// TIA Portal V19 export
DATA_BLOCK "AreaGen_Msg_Alarms"   // DB181
// stored: InstanceOfName MsgManager, InstanceOfType FB
"MsgManager"
   // VAR_INPUT
   //    Ack : Bool;
   // END_VAR
   // VAR_OUTPUT
   //    MessagePresence : Bool;
   //    NewMessage : Bool;
   //    MessageCount : Int;
   // END_VAR
   // VAR_IN_OUT
   //    Messages : Array[*] of Bool;
   //    MessagesHMI : Array[*] of Word;
   //    MessagesACK : Array[*] of Word;
   // END_VAR
   // VAR
   //    MsgDim : DInt;
   //    HmiMsgDim : DInt;
   //    AckMsgDim : DInt;
   //    MsgCount : Int;
   //    Status : Int;
   //    IndexBuild : Int;
   //    IndexCompare : Int;
   //    LoopStart : Int;
   //    LoopEnd : Int;
   //    HMIIndex : Int;
   //    CompareWord : Word;
   //    "A" : Word;
   //    MvBlkVar_ErrorID : Int;
   // END_VAR
BEGIN
END_DATA_BLOCK
